// TIA Portal V17 export
// export: Created 2024-09-02T12:50:24.1458979Z, ExportSetting WithDefaults, DisplayName Totally Integrated Automation Portal, DisplayVersion V17, DisplayName TIA Portal Openness, DisplayVersion V17, DisplayName TIA Portal Version Control Interface, DisplayVersion V17, DisplayName STEP 7 Professional, DisplayVersion V17, DisplayName STEP 7 Safety, DisplayVersion V17, DisplayName WinCC Professional, DisplayVersion V17
DATA_BLOCK "DB_MES_Settings_OP70"   // DB601
{ S7_Optimized_Access := 'TRUE' }
VERSION : 0.1
// stored: AutoNumber false, DBAccessibleFromOPCUA true, IsOnlyStoredInLoadMemory false, IsRetainMemResEnabled false, IsWriteProtectedInAS false, MemoryReserve 100
   VAR RETAIN
      HMI : Struct   // HMI structure
         MesMainButton : "UDT_MES_Button";   // Main button on template screen
         MesApproveButton { S7_SetPoint := 'True'} : "UDT_MES_Button";   // Approve button for reason of MES deselection
         MesActivationButton { S7_SetPoint := 'True'} : "UDT_MES_Button";   // Button for reset of MES deselection
         OptionActivated : USInt;   // Option activated
         DeselectionOption { S7_SetPoint := 'True'} : USInt;   // Deselection option
      END_STRUCT;
   END_VAR
   VAR
      DeselectionOption : Array[0..4] of String[15];   // Array of deselection options
   END_VAR
   VAR RETAIN
      EDGE : Array[0..7] of Bool;   // HLP Edge
      MesDeselected : Bool;   // MES deselection bit
   END_VAR
   VAR
      MES_Error_ACK : Bool;
      PopUp_Start : Bool;
      Time_stamp_start_70_1 : Bool;
      Time_stamp_stop_70_1 : Bool;
      Time_stamp_start_70_2 : Bool;
      Time_stamp_stop_70_2 : Bool;
      Time_stamp_start_70_3 : Bool;
      Time_stamp_stop_70_3 : Bool;
      StationState : Array[0..15] of Bool;
      StationState_Word : Word;
   END_VAR
BEGIN
   DeselectionOption[1] := 'Golden_Part';
   DeselectionOption[2] := 'Maintenance';
   DeselectionOption[3] := 'MSA';
   DeselectionOption[4] := 'Test_Purposes';
END_DATA_BLOCK
